Fanuc KAREL source: kc00041.KL

-- PROVISIONAL review KL for V940-1; original PC SHA256 52842232d1268c529253f68a058097e3fda050f2cc44745009aad5f17a215f7f
-- Incomplete behavior may be omitted. Consult companion uncertainty JSON. Do not deploy.
PROGRAM KC00041
%NOLOCKGROUP
BEGIN
  -- V9_ZERO_TABLE_METADATA_HINT layout=0002_ascii; no indexed target words; source/name/runtime held
  -- UNRESOLVED_PC offsets 5-33; opcodes 27,22,22,22,22,31
  -- UNRESOLVED_PC offsets 38-42; opcodes 7F
END KC00041
